Fanuc KAREL source: kd00031.KL

PROGRAM KD00031
%STACKSIZE=65535
%PRIORITY=65535
%NOLOCKGROUP
VAR
I : INTEGER
J : INTEGER
B : BOOLEAN
R : REAL
S : STRING[80]
BEGIN
-- UNRESOLVED_PC line 10 opcodes [9D 81 18 9C 12 22 9D 13 04] marker_code=0
END KD00031
